{attribute 'qualified_only'}
VAR_GLOBAL
	loop: MyWorker;
END_VAR

(* stored: Version 1.1.0.1
   GVL SharedWorker: Id {d7fae350-a1e5-4b5c-83b3-cdb58505f079} *)
